FUNCTION_BLOCK gain_min1 (* Basic FB with empty ECC *)
  (* Standard: 61499-2 *)
  (* Version 1.0, 2021-03-30, Lenovo *)
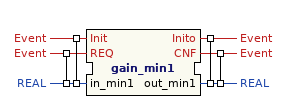
  EVENT_INPUT
    Init WITH in_min1;
    REQ WITH in_min1;
  END_EVENT
  EVENT_OUTPUT
    Inito WITH out_min1;
    CNF WITH out_min1;
  END_EVENT
  VAR_INPUT
    in_min1 : REAL;
  END_VAR
  VAR_OUTPUT
    out_min1 : REAL;
  END_VAR
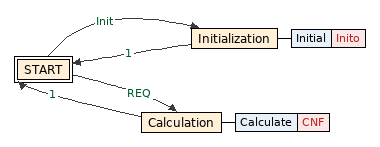
  EC_STATES
    START; (* Initial State *)
    Initialization : Initial -> Inito;
    Calculation : Calculate -> CNF;
  END_STATES
  EC_TRANSITIONS
    START TO Initialization := Init;
    Initialization TO START := 1;
    START TO Calculation := REQ;
    Calculation TO START := 1;
  END_TRANSITIONS
  ALGORITHM Initial IN ST: (* New Algorithm *)

  END_ALGORITHM
  ALGORITHM Calculate IN ST: (* New Algorithm *)
out_min1:=(-0.1)*in_min1;
  END_ALGORITHM
END_FUNCTION_BLOCK
